# EPICS substitutions: CsHeaterApp/Db/Watlow_PM_Monitor.substitutions
file Watlow_PM_Monitor.template
{
pattern {  s, ta,      ss, mod, ch, CMA, hPr, CPr, PvA, CLS, AtS}
        { '', SE,  Watlow,   1,  1,   0,   0,   2,  42,   0,   4}
        { '', SE,  Watlow,   1,  2,   0,   0,   2,  42,   0,   4}
}
